TYPE "生产线to上位机"
VERSION : 0.1
   STRUCT
      产线状态 : Struct
         "1秒心跳" : Bool;   // 每秒一次脉冲信号，用于判断通信情况
         手动模式 : Bool;
         自动模式 : Bool;
         运行状态 : Bool;
         "4" : Bool;
         "5" : Bool;
         "6" : Bool;
         "7" : Bool;
         "8" : Bool;
         "9" : Bool;
         "10" : Bool;
         "11" : Bool;
         "12" : Bool;
         "13" : Bool;
         "14" : Bool;
         "15" : Bool;
      END_STRUCT;
      包装机 : Struct
         包装机状态 : Int;   // 0通信中断，1=待机中，2=生成中，其他=异常
         申请读码 : Int;   // 1=申请读码
         袋码数据 : String[32];   // 字符串
         包装重量 : Real;
         包装时间 : Real;
      END_STRUCT;
      称重机 : Struct
         称重机状态 : Int;   // 0通信中断，1=待机中，2=生成中，其他=异常
         申请读码 : Int;   // 1=申请读码
         袋码数据 : String[32];   // 字符串
         称重重量 : Real;   // 重量 单位：kg
      END_STRUCT;
      喷码机 : Struct
         喷码机状态 : Int;   // 0通信中断，1=待机中，2=生成中，其他=异常
         申请读码 : Int;   // 1=申请读码
         袋码数据 : String[32];   // 字符串
      END_STRUCT;
      码垛 : Struct
         码垛机状态 : Int;
         申请读码 : Int;   // 1=申请读码
         码垛袋码 : String[32];   // 袋码信息
         码垛包数 : Int;   // 实时包数
      END_STRUCT;
      组托 : Struct
         申请读码 : Int;   // 1=申请读码
         袋码数据 : String[32];
         垛盘码数据 : String[32];
      END_STRUCT;
      缠绕覆膜 : Struct
         申请读码 : Int;   // 1=申请读码
         袋码数据 : String[32];
      END_STRUCT;
      贴标 : Struct
         申请读码 : Int;   // 1=申请读码
         袋码数据 : String[32];
         垛盘码数据 : String[32];
      END_STRUCT;
   END_STRUCT;

END_TYPE

DATA_BLOCK "1002输送to上位机"
{ S7_Optimized_Access := 'FALSE' }
VERSION : 0.1
NON_RETAIN
   STRUCT
      to上位机 { S7_SetPoint := 'False'} : "生产线to上位机";
   END_STRUCT;


BEGIN

END_DATA_BLOCK

